Staubli VAL3: Robot_pippeting.pjx

--- Robot_pippeting.pjx ---
Parameters version=s8.8.3cs9_BS1660 stackSize=200000 millimeterUnit=true
Program file=ComPlc.pgx
Program file=Control.pgx
Program file=Emergencia.pgx
Program file=Init.pgx
Program file=Log.pgx
Program file=N10_AproBanyera.pgx
Program file=N11_Banyera.pgx
Program file=N12_AproAmpolla.pgx
Program file=N13_Ampolla.pgx
Program file=N15_AproAgafarPuntes.pgx
Program file=N16_AgafarPuntes.pgx
Program file=N17_AproTirarPuntes.pgx
Program file=N18_TirarPuntes.pgx
Program file=N1_Home.pgx
Program file=N20_AproDosi.pgx
Program file=N21_Dosi.pgx
Program file=N22_PosDosi.pgx
Program file=Principal.pgx
Program file=Safety.pgx
Program file=Supervision.pgx
Program file=start.pgx
Program file=stop.pgx
Data file=Robot_pippeting.dtx

--- Robot_pippeting.dtx ---
aio aiAngleInclinarPipieta = {link=E954DA08-7D0C-47C0-8458-4D7DB0686071}
aio aiNumAmpolla = {link=F94C03B3-E86B-41EA-9D21-23C2AFB25672}
aio aiNumBanyera = {link=3DE16CC9-CC25-4818-8F3E-A7F806CB7947}
aio aiNumPipeta = {link=5259214B-6548-4F3D-A189-73563EE6598D}
aio aiNumPlacaDosi = {link=C4FBE503-E51F-4D58-BE10-749D221ACEB2}
aio aiProgramaPlc = {link=8E5652B8-E4D3-4267-ADD0-9C5A815DF2D8}
aio aiWordComPlc = {link=5C2A04D3-4005-4B43-8647-C0FC7B49D3AE}
aio aiXOffset = {link=95067B68-557B-4170-88AF-FC9CF5B8ED7A}
aio aiYOffset = {link=396181D2-5171-4A97-9799-32514BBB5F95}
aio aiZApro = {link=2D158B67-9924-4741-B554-50FB73F41045}
aio aiZOffset = {link=7513B562-B4FE-4098-AA1C-29A8706B731C}
aio aoForceJ1 = {link=9B11B2FE-99BA-4B55-9ED8-E4037A61E514}
aio aoForceJ2 = {link=DFC528C5-C573-4C02-A89E-35D8A1151078}
aio aoForceJ3 = {link=EC117CCB-E5D8-4A5C-AB6E-61FBA1760A17}
aio aoForceJ4 = {link=24340562-5DCA-47E3-A269-832024611405}
aio aoForceJ5 = {link=DB01A7CB-9BAD-4D46-B614-A585779504D9}
aio aoForceJ6 = {link=7A496CE7-D747-4637-B99A-202C76C7E7CC}
aio aoProgramaRobot = {link=5113B9A1-604C-4D8B-9163-7217CBF800C7}
aio aoStatusRobot = {link=F45B1EFD-4428-4D7D-8172-ECCCA511584C}
aio aoTascaAlarma = {link=53CEF201-0BB5-4BE1-8271-49FFF55CF52D}
aio aoWordComRobot = {link=6DF138BB-5CBA-4ACE-9C62-0AC3DF2353CB}
aio aoWorkingMode = {link=F7E03293-48A3-4B69-9598-2FE8DDFE0186}
aio aoXActual = {link=7FC267A8-BFA4-4039-BDA4-9FB4B4F71D48}
aio aoYActual = {link=E23CA4B2-A08C-4C00-8E97-94551E73BB09}
aio aoZActual = {link=78A73075-60CA-4FDB-AFF0-231125481CE1}
aio aoZonaHome = {link=F5709703-FBB2-4816-9A2C-2FC6F0D8F434}
bool bNewLog
bool bPrimerCicle
bool bTaskDone
dio diAlarmaPlc = {link=E7921EDF-610C-4E3F-84A7-2F1F4421B713}
dio diMarxaMaquina = {link=C1F67030-A9C1-420C-9B9B-1F49F7080557}
dio diSafetyRearme = {link=5367EF22-1F58-447B-AD12-D8B84F185C6B}
dio doAlarmaColisioRobot = {link=EA8AD671-7535-4BE0-BEBB-B9246DF094E3}
dio doAlarmaTascaRobot = {link=FCAEE04F-32B9-421A-B1DD-A8CEAA94D1C9}
dio doRobotEnMoviment = {link=B70DA9EE-8DF7-4C99-91DF-7149F2D942A3}
dio doRobotHome = {link=9957E281-FF01-4081-BA5E-7A249685580C}
dio doRobotPreparat = {link=19F8D819-A10B-480E-B6CD-15D2D35E2133}
dio doTaskDone = {link=0B0F13F6-DB8F-450C-AEE5-782BE1039C53}
frame fTaula = {fatherId=world[0]}
jointRx jHome = {j1=-3.455563, j2=6.0127238, j3=105.394535, j4=0.000031955, j5=68.591721, j6=-183.446968}
mdesc mAgafarPuntes = {accel=10, vel=10, decel=10, leave=0, reach=0}
mdesc mHome = {accel=25, vel=25, decel=25, leave=0, reach=0}
mdesc mLent = {accel=25, vel=25, decel=25, leave=10, reach=10}
mdesc mMig = {accel=50, vel=50, decel=50}
mdesc mNomSpeed
num nAngleInclinarPipeta
num nInerciaEina[3 3]
  [0,0] = 0.284
  [1,1] = 0.348
  [2,2] = 0.212
num nJointForce[6]
  [0] = 1.760942
  [1] = -21.676362
  [2] = -3.171848
  [3] = 1.641233
  [4] = -2.820579
  [5] = -0.389449
num nLog
num nPesEina = 15.8
num nSeqHome
num nWordComRobot = 6190
num nXOffset
num nYOffset
num nZApro = 50
num nZOffset
pointRx pAgafarPuntes1 = {x=287.432018, y=270.157151, z=-382.0291842, rx=179.996843, ry=-0.00380694, rz=0.700516, shoulder=lefty, elbow=epositive, wrist=wpositive, fatherId=fTaula[0]}
pointRx pAgafarPuntes8 = {x=285.860304, y=302.266054, z=-361.378441, rx=179.997149, ry=-0.00370527, rz=0.700442, shoulder=lefty, elbow=epositive, wrist=wpositive, fatherId=fTaula[0]}
pointRx pAmpolla[3]
  [0] = {x=493.522667, y=144.0778037, z=-386.621607, rx=179.997388, ry=-0.00407881, rz=0.700451, shoulder=lefty, elbow=epositive, wrist=wpositive, fatherId=fTaula[0]}
  [1] = {x=493.522667, y=144.0778037, z=-386.621607, rx=179.997388, ry=-0.00407881, rz=0.700451, shoulder=lefty, elbow=epositive, wrist=wpositive, fatherId=fTaula[0]}
  [2] = {x=546.605553, y=142.888702, z=-386.0523536, rx=179.997158, ry=-0.00493572, rz=0.700473, shoulder=lefty, elbow=epositive, wrist=wpositive, fatherId=fTaula[0]}
pointRx pBanyera[3]
  [0] = {x=336.466109, y=102.428458, z=-384.993166, rx=-0.00440943, ry=-179.995824, rz=-89.890495, shoulder=lefty, elbow=epositive, wrist=wpositive, fatherId=fTaula[0]}
  [1] = {x=336.466109, y=102.428458, z=-384.993166, rx=-0.00440943, ry=-179.995824, rz=-89.890495, shoulder=lefty, elbow=epositive, wrist=wpositive, fatherId=fTaula[0]}
  [2] = {x=336.466107, y=182.839383, z=-384.995018, rx=-0.003849, ry=-179.995539, rz=-89.890699, shoulder=lefty, elbow=epositive, wrist=wpositive, fatherId=fTaula[0]}
pointRx pDosi1[4]
  [0] = {x=305.52358, y=28.950334, z=-381.105899, rx=-0.00502749, ry=-179.983412, rz=-88.969574, shoulder=lefty, elbow=epositive, wrist=wpositive, fatherId=fTaula[0]}
  [1] = {x=305.523534, y=28.950368, z=-381.105899, rx=-0.00502365, ry=-179.983406, rz=-88.969579, shoulder=lefty, elbow=epositive, wrist=wpositive, fatherId=fTaula[0]}
  [2] = {x=306.96586, y=-130.963134, z=-381.122863, rx=-0.00532463, ry=-179.983113, rz=-88.9695, shoulder=lefty, elbow=epositive, wrist=wpositive, fatherId=fTaula[0]}
  [3] = {x=307.512874, y=-290.507285, z=-381.117547, rx=-0.00478912, ry=-179.98278, rz=-88.969551, shoulder=lefty, elbow=epositive, wrist=wpositive, fatherId=fTaula[0]}
pointRx pDosi8[4]
  [0] = {x=337.355483, y=31.174712, z=-385.0727918, rx=-0.0019009, ry=-179.993411, rz=-88.962152, shoulder=lefty, elbow=epositive, wrist=wpositive, fatherId=fTaula[0]}
  [1] = {x=337.355483, y=31.174712, z=-385.0727918, rx=-0.0019009, ry=-179.993411, rz=-88.962152, shoulder=lefty, elbow=epositive, wrist=wpositive, fatherId=fTaula[0]}
  [2] = {x=338.549957, y=-128.589669, z=-385.0544196, rx=0.000914256, ry=-179.993163, rz=-88.965193, shoulder=lefty, elbow=epositive, wrist=wpositive, fatherId=fTaula[0]}
  [3] = {x=339.326592, y=-288.609993, z=-385.0722156, rx=0.00206439, ry=-179.994818, rz=-88.964134, shoulder=lefty, elbow=epositive, wrist=wpositive, fatherId=fTaula[0]}
pointRx pHereHome = {x=172.623152, y=-333.816468, z=-286.331237, rx=0.00171927, ry=-179.997666, rz=-88.962057, shoulder=lefty, elbow=epositive, wrist=wpositive, fatherId=fTaula[0]}
pointRx pHome = {x=319.622111, y=0.736493, z=-179.743756, rx=180, shoulder=lefty, elbow=epositive, wrist=wpositive, fatherId=fTaula[0]}
pointRx pTirarPuntes = {x=172.623152, y=-333.816468, z=-336.331237, rx=0.00171927, ry=-179.997666, rz=-88.962057, shoulder=lefty, elbow=epositive, wrist=wpositive, fatherId=fTaula[0]}
string sLog[50]
  [1] = "1 - Inici: HOME"
  [2] = "17 - Fi: ANAR A APRO TIRAR PUNTES"
  [3] = "17 - Inici: ANAR A APRO TIRAR PUNTES"
  [4] = "18 - Fi: ANAR A TIRAR PUNTES"
  [5] = "18 - Inici: ANAR A TIRAR PUNTES"
  [6] = "17 - Fi: ANAR A APRO TIRAR PUNTES"
  [7] = "17 - Inici: ANAR A APRO TIRAR PUNTES"
  [8] = "20 - Fi: ANAR A APRO DOSI"
  [9] = "20 - Inici: ANAR A APRO DOSI"
  [10] = "22 - Fi: ANAR A POSICIONAT DOSI"
  [11] = "22 - Inici: ANAR A POSICIONAT DOSI"
  [12] = "21 - Fi: ANAR A DOSI"
  [13] = "21 - Inici: ANAR A DOSI"
  [14] = "20 - Fi: ANAR A APRO DOSI"
  [15] = "20 - Inici: ANAR A APRO DOSI"
  [16] = "20 - Fi: ANAR A APRO DOSI"
  [17] = "20 - Inici: ANAR A APRO DOSI"
  [18] = "22 - Fi: ANAR A POSICIONAT DOSI"
  [19] = "22 - Inici: ANAR A POSICIONAT DOSI"
  [20] = "21 - Fi: ANAR A DOSI"
  [21] = "21 - Inici: ANAR A DOSI"
  [22] = "20 - Fi: ANAR A APRO DOSI"
  [23] = "20 - Inici: ANAR A APRO DOSI"
  [24] = "20 - Fi: ANAR A APRO DOSI"
  [25] = "20 - Inici: ANAR A APRO DOSI"
  [26] = "21 - Fi: ANAR A DOSI"
  [27] = "21 - Inici: ANAR A DOSI"
  [28] = "20 - Fi: ANAR A APRO DOSI"
  [29] = "20 - Inici: ANAR A APRO DOSI"
  [30] = "15 - Fi: ANAR A APRO AGAFAR PUNTES"
  [31] = "15 - Inici: ANAR A APRO AGAFAR PUNTES"
  [32] = "16 - Fi: ANAR A AGAFAR PUNTES"
  [33] = "16 - Inici: ANAR A AGAFAR PUNTES"
  [34] = "15 - Fi: ANAR A APRO AGAFAR PUNTES"
  [35] = "15 - Inici: ANAR A APRO AGAFAR PUNTES"
  [36] = "17 - Fi: ANAR A APRO TIRAR PUNTES"
  [37] = "17 - Inici: ANAR A APRO TIRAR PUNTES"
  [38] = "18 - Fi: ANAR A TIRAR PUNTES"
  [39] = "18 - Inici: ANAR A TIRAR PUNTES"
  [40] = "17 - Fi: ANAR A APRO TIRAR PUNTES"
  [41] = "17 - Inici: ANAR A APRO TIRAR PUNTES"
  [42] = "20 - Fi: ANAR A APRO DOSI"
  [43] = "20 - Inici: ANAR A APRO DOSI"
  [44] = "22 - Fi: ANAR A POSICIONAT DOSI"
  [45] = "22 - Inici: ANAR A POSICIONAT DOSI"
  [46] = "21 - Fi: ANAR A DOSI"
  [47] = "21 - Inici: ANAR A DOSI"
  [48] = "20 - Fi: ANAR A APRO DOSI"
  [49] = "20 - Inici: ANAR A APRO DOSI"
string sNewLog = "1 - Fi: HOME"
tool tToolActiva = {z=285, fatherId=flange[0]}
tool tToolPipeta1 = {z=300, fatherId=flange[0]}
tool tToolPipeta8 = {z=285, fatherId=flange[0]}
trsf trEina = {x=94.8, y=-0.4, z=220.5}

--- start.pgx ---
program start()
begin

  taskCreate "Supervision",50,Supervision()
  taskCreate "ComPlc",50,ComPlc()
  taskCreate "Init",50,Init()

  // Mostrar pantalla d'usuari
  userPage("main")
end

--- ComPlc.pgx ---
program ComPlc()
begin
  do
    // Word de vida de la comunicació entre el robot i el PLC
    if nWordComRobot>10000
      nWordComRobot=0
    endIf
    nWordComRobot=nWordComRobot+1
    aioSet(aoWordComRobot,nWordComRobot)

  until false
end

--- Control.pgx ---
program Control()
  local pointRx l_pHere
begin
  do
    // Status robot
    aioSet(aoStatusRobot,esStatus())
    aioSet(aoWorkingMode,workingMode())

    // Velocitat del robot segons hmi
    //setMonitorSpeed(aioGet(aiVelocitatRobot))

    // Donar potencia al robot
    if esStatus()==0 and diAlarmaPlc==false and isPowered()==false and workingMode()==4
      enablePower()
    endIf

    // Definir tool de treball
    if aioGet(aiNumPipeta)==2
      tToolActiva=tToolPipeta8
    else
      tToolActiva=tToolPipeta1
    endIf

    // Envelope error - Alarma possible colisió del robot
    //doAlarmaColisioRobot=$envelopeError()

    // Error "Posició cartesiana fóra de límits"
    if taskStatus("Principal")==531 or taskStatus("N1_Home")==531 or taskStatus("N10_AproBanyera")==531 or taskStatus("N11_Banyera")==531 or taskStatus("N15_AproAgafarPuntes")==531 or taskStatus("N16_AgafarPuntes")==531 or taskStatus("N17_AproTirarPuntes")==531 or taskStatus("N18_TirarPuntes")==531 or taskStatus("N20_AproDosi")==531 or taskStatus("N21_Dosi")==531 or taskStatus("N22_PosDosi")==531 or taskStatus("N12_AproAmpolla")==531 or taskStatus("N13_Ampolla")==531
      aioSet(aoTascaAlarma,aioGet(aoProgramaRobot))
      doAlarmaTascaRobot=true
    else
      doAlarmaTascaRobot=false
    endIf

    // Enviar al PLC la força de cada motor del robot (Nm)
    getJointForce(nJointForce)
    aioSet(aoForceJ1,nJointForce[0])
    aioSet(aoForceJ2,nJointForce[1])
    aioSet(aoForceJ3,nJointForce[2])
    aioSet(aoForceJ4,nJointForce[3])
    aioSet(aoForceJ5,nJointForce[4])
    aioSet(aoForceJ6,nJointForce[5])

    // Enviar al PLC la posició actual del robot
    l_pHere=here(tToolActiva,world)
    aioSet(aoXActual,l_pHere.trsf.x)
    aioSet(aoYActual,l_pHere.trsf.y)
    aioSet(aoZActual,l_pHere.trsf.z)

  until false
end

--- Emergencia.pgx ---
program Emergencia()
begin

  do
    if diAlarmaPlc==true

      taskKill("Principal")
      taskKill("N1_Home")
      taskKill("N10_AproBanyera")
      taskKill("N11_Banyera")
      taskKill("N12_AproAmpolla")
      taskKill("N13_Ampolla")
      taskKill("N15_AproAgafarPuntes")
      taskKill("N16_AgafarPuntes")
      taskKill("N17_AproTirarPuntes")
      taskKill("N18_TirarPuntes")
      taskKill("N20_AproDosi")
      taskKill("N21_Dosi")
      taskKill("N22_PosDosi")


      resetMotion()
      //Reset variables
      doRobotHome=false
      doRobotEnMoviment=false

      doAlarmaColisioRobot=false
      doTaskDone=false

      bTaskDone=false
      bPrimerCicle=false
      nSeqHome=0
      aioSet(aoProgramaRobot,0)
      aioSet(aoZonaHome,0)

      wait(diAlarmaPlc==false)

      taskCreate "Principal",50,Principal()
    endIf
    delay(0)
  until false


end

--- Init.pgx ---
program Init()
begin


  // Inicialització de variables
  doRobotHome=false
  doRobotEnMoviment=false
  doRobotPreparat=false
  doAlarmaColisioRobot=false
  doAlarmaTascaRobot=false
  doTaskDone=false
  bTaskDone=false
  bPrimerCicle=false
  bNewLog=false
  sLog=""
  nSeqHome=0
  aioSet(aoProgramaRobot,0)
  aioSet(aoZonaHome,0)
  nAngleInclinarPipeta=0

  //  // Definir l'eina (valores de inercia en kg·m2)
  nInerciaEina[0,0]=0.284
  nInerciaEina[0,1]=0
  nInerciaEina[0,2]=0
  nInerciaEina[1,0]=0
  nInerciaEina[1,1]=0.348
  nInerciaEina[1,2]=0
  nInerciaEina[2,0]=0
  nInerciaEina[2,1]=0
  nInerciaEina[2,2]=0.212
  trEina={94.8,-0.4,220.5,0,0,0}
  nPesEina=15.8
  setPayload(flange,nPesEina,trEina,nInerciaEina)


  doRobotPreparat=true

  taskCreate "Control",50,Control()
  taskCreate "Log",50,Log()
  taskCreate "Safety",50,Safety()
  taskCreate "Principal",50,Principal()
  taskCreate "Emergencia",2,Emergencia()

end

--- Log.pgx ---
program Log()
begin
  do
    // Registrar un nou event al logger
    if bNewLog==true
      // Desplaçar registre d'events
      for nLog=49 to 1 step -1
        sLog[nLog]=sLog[nLog-1]
      endFor
      // Afegir nou event
      sLog[0]=sNewLog
      bNewLog=false
    endIf

  until false
end

--- N10_AproBanyera.pgx ---
program N10_AproBanyera()
  local pointRx l_pAproBanyera
begin

  // Anar a l'aproximació del punt d'agafar líquid de la banyera
  l_pAproBanyera=pBanyera[aioGet(aiNumBanyera)]
  l_pAproBanyera.trsf.x=l_pAproBanyera.trsf.x+nXOffset
  l_pAproBanyera.trsf.y=l_pAproBanyera.trsf.y+nYOffset
  l_pAproBanyera.trsf.z=l_pAproBanyera.trsf.z+nZOffset

  if nZApro>0
    l_pAproBanyera.trsf.z=l_pAproBanyera.trsf.z+nZApro
  else
    l_pAproBanyera.trsf.z=l_pAproBanyera.trsf.z+100
  endIf

  movel(l_pAproBanyera,tToolActiva,mLent)
  waitEndMove()

  bTaskDone=true
end

--- N11_Banyera.pgx ---
program N11_Banyera()
  local pointRx l_pBanyera
begin

  // Anar al punt de la banyera
  l_pBanyera=pBanyera[aioGet(aiNumBanyera)]
  l_pBanyera.trsf.x=l_pBanyera.trsf.x+nXOffset
  l_pBanyera.trsf.y=l_pBanyera.trsf.y+nYOffset
  l_pBanyera.trsf.z=l_pBanyera.trsf.z+nZOffset
  movel(l_pBanyera,tToolActiva,mLent)
  waitEndMove()

  bTaskDone=true
end

--- N12_AproAmpolla.pgx ---
program N12_AproAmpolla()
  local pointRx l_pAproAmpolla
begin

  // Anar a l'aproximació del punt d'agafar líquid de l'ampolla
  l_pAproAmpolla=pAmpolla[aioGet(aiNumAmpolla)]
  l_pAproAmpolla.trsf.x=l_pAproAmpolla.trsf.x+nXOffset
  l_pAproAmpolla.trsf.y=l_pAproAmpolla.trsf.y+nYOffset
  l_pAproAmpolla.trsf.z=l_pAproAmpolla.trsf.z+nZOffset

  if nZApro>0
    l_pAproAmpolla.trsf.z=l_pAproAmpolla.trsf.z+nZApro
  else
    l_pAproAmpolla.trsf.z=l_pAproAmpolla.trsf.z+100
  endIf

  movel(l_pAproAmpolla,tToolActiva,mLent)
  waitEndMove()

  bTaskDone=true
end

--- N13_Ampolla.pgx ---
program N13_Ampolla()
  local pointRx l_pAmpolla
begin

  // Anar al punt de l'ampolla
  l_pAmpolla=pAmpolla[aioGet(aiNumAmpolla)]
  l_pAmpolla.trsf.x=l_pAmpolla.trsf.x+nXOffset
  l_pAmpolla.trsf.y=l_pAmpolla.trsf.y+nYOffset
  l_pAmpolla.trsf.z=l_pAmpolla.trsf.z+nZOffset
  movel(l_pAmpolla,tToolActiva,mLent)
  waitEndMove()

  bTaskDone=true
end

--- N15_AproAgafarPuntes.pgx ---
program N15_AproAgafarPuntes()
  local pointRx l_pAproAgafarPuntes
begin

  // Anar a l'aproximació del punt d'agafar puntes
  if aioGet(aiNumPipeta)==2
    l_pAproAgafarPuntes=pAgafarPuntes8
  else
    l_pAproAgafarPuntes=pAgafarPuntes1
  endIf

  l_pAproAgafarPuntes.trsf.x=l_pAproAgafarPuntes.trsf.x+nXOffset
  l_pAproAgafarPuntes.trsf.y=l_pAproAgafarPuntes.trsf.y+nYOffset
  l_pAproAgafarPuntes.trsf.z=l_pAproAgafarPuntes.trsf.z+nZOffset

  if nZApro>0
    l_pAproAgafarPuntes.trsf.z=l_pAproAgafarPuntes.trsf.z+nZApro
  else
    l_pAproAgafarPuntes.trsf.z=l_pAproAgafarPuntes.trsf.z+100
  endIf

  movel(l_pAproAgafarPuntes,tToolActiva,mLent)
  waitEndMove()

  bTaskDone=true
end

--- N16_AgafarPuntes.pgx ---
program N16_AgafarPuntes()
  local pointRx l_pAgafarPuntes
  local pointRx l_pAgafarPuntesRapid
begin

  // Anar al punt de la banyera
  if aioGet(aiNumPipeta)==2
    l_pAgafarPuntes=pAgafarPuntes8
  else
    l_pAgafarPuntes=pAgafarPuntes1
  endIf

  l_pAgafarPuntes.trsf.x=l_pAgafarPuntes.trsf.x+nXOffset
  l_pAgafarPuntes.trsf.y=l_pAgafarPuntes.trsf.y+nYOffset
  l_pAgafarPuntes.trsf.z=l_pAgafarPuntes.trsf.z+nZOffset
  l_pAgafarPuntesRapid=l_pAgafarPuntes
  l_pAgafarPuntesRapid.trsf.z=l_pAgafarPuntesRapid.trsf.z+20
  movel(l_pAgafarPuntesRapid,tToolActiva,mLent)
  waitEndMove()
  movel(l_pAgafarPuntes,tToolActiva,mAgafarPuntes)
  waitEndMove()

  bTaskDone=true
end

--- N17_AproTirarPuntes.pgx ---
program N17_AproTirarPuntes()
  local pointRx l_pAproTirarPuntes
begin

  // Anar a l'aproximació del punt de tirar puntes
  l_pAproTirarPuntes=pTirarPuntes
  l_pAproTirarPuntes.trsf.x=l_pAproTirarPuntes.trsf.x+nXOffset
  l_pAproTirarPuntes.trsf.y=l_pAproTirarPuntes.trsf.y+nYOffset
  l_pAproTirarPuntes.trsf.z=l_pAproTirarPuntes.trsf.z+nZOffset

  if nZApro>0
    l_pAproTirarPuntes.trsf.z=l_pAproTirarPuntes.trsf.z+nZApro
  else
    l_pAproTirarPuntes.trsf.z=l_pAproTirarPuntes.trsf.z+50
  endIf

  movel(l_pAproTirarPuntes,tToolActiva,mLent)
  waitEndMove()

  bTaskDone=true
end

--- N18_TirarPuntes.pgx ---
program N18_TirarPuntes()
  local pointRx l_pTirarPuntes
begin

  // Anar al punt de tirar puntes
  l_pTirarPuntes=pTirarPuntes
  l_pTirarPuntes.trsf.x=l_pTirarPuntes.trsf.x+nXOffset
  l_pTirarPuntes.trsf.y=l_pTirarPuntes.trsf.y+nYOffset
  l_pTirarPuntes.trsf.z=l_pTirarPuntes.trsf.z+nZOffset
  movel(l_pTirarPuntes,tToolActiva,mLent)
  waitEndMove()

  bTaskDone=true
end

--- N1_Home.pgx ---
program N1_Home()
  local pointRx l_pHere
begin
  do

    switch nSeqHome

      // Inici de la seqüència
      case 0
        // Anar a home
        doRobotHome=false
        doRobotEnMoviment=true
        aioSet(aoZonaHome,0)
        waitEndMove()
        // Comprovar a quina posició es troba el robot
        l_pHere=here(tToolActiva,fTaula)
        pHereHome=l_pHere
        nSeqHome=10
      break

      // Pujar verticalment fins a una cota segura en Z
      case 10
        if l_pHere.trsf.z<pHome.trsf.z
          l_pHere.trsf.z=pHome.trsf.z
          movel(l_pHere,tToolActiva,mHome)
          waitEndMove()
          nSeqHome=20
        else
          nSeqHome=20
        endIf
      break

      // Comprovar on es troba el robot
      case 20
        // Ja està en posició de Home
        aioSet(aoZonaHome,99)
        nSeqHome=1000
      break

      // Fi del HOME
      case 1000
        movel(pHome,tToolActiva,mHome)
        waitEndMove()
        doRobotHome=true
        doRobotEnMoviment=false
        bTaskDone=true
        nSeqHome=1001
      break
    endSwitch
  until nSeqHome==1001
end

--- N20_AproDosi.pgx ---
program N20_AproDosi()
  local pointRx l_pAproDosi
begin

  // Anar a l'aproximació vertical de dosificar placa
  if aioGet(aiNumPipeta)==2
    l_pAproDosi=pDosi8[aioGet(aiNumPlacaDosi)]
  else
    l_pAproDosi=pDosi1[aioGet(aiNumPlacaDosi)]
  endIf

  l_pAproDosi.trsf.x=l_pAproDosi.trsf.x+nXOffset
  l_pAproDosi.trsf.y=l_pAproDosi.trsf.y+nYOffset
  l_pAproDosi.trsf.z=l_pAproDosi.trsf.z+nZOffset

  if nZApro>0
    l_pAproDosi.trsf.z=l_pAproDosi.trsf.z+nZApro
  else
    l_pAproDosi.trsf.z=l_pAproDosi.trsf.z+25
  endIf

  l_pAproDosi.trsf.rx=l_pAproDosi.trsf.rx+aioGet(aiAngleInclinarPipieta)

  movel(l_pAproDosi,tToolActiva,mLent)
  waitEndMove()

  bTaskDone=true
end

--- N21_Dosi.pgx ---
program N21_Dosi()
  local pointRx l_pDosi
begin

  // Anar al punt de dosificar placa
  if aioGet(aiNumPipeta)==2
    l_pDosi=pDosi8[aioGet(aiNumPlacaDosi)]
  else
    l_pDosi=pDosi1[aioGet(aiNumPlacaDosi)]
  endIf
  l_pDosi.trsf.x=l_pDosi.trsf.x+nXOffset
  l_pDosi.trsf.y=l_pDosi.trsf.y+nYOffset
  l_pDosi.trsf.z=l_pDosi.trsf.z+nZOffset
  l_pDosi.trsf.rx=l_pDosi.trsf.rx+aioGet(aiAngleInclinarPipieta)

  movel(l_pDosi,tToolActiva,mLent)
  waitEndMove()

  bTaskDone=true
end

--- N22_PosDosi.pgx ---
program N22_PosDosi()
  local pointRx l_pDosi
begin

  // Moure puntes per treure les gotes
  l_pDosi=here(tToolActiva,fTaula)
  l_pDosi.trsf.x=l_pDosi.trsf.x+nXOffset
  l_pDosi.trsf.y=l_pDosi.trsf.y+nYOffset
  l_pDosi.trsf.z=l_pDosi.trsf.z+nZOffset
  movel(l_pDosi,tToolActiva,mLent)
  waitEndMove()

  bTaskDone=true
end

--- Principal.pgx ---
program Principal()
begin
  do

    // Esperar aiProgramaPlc <> 0
    do
      delay(0)
    until (aioGet(aiProgramaPlc)!=0)

    // Processar X,Y,Z offset posició
    nXOffset=aioGet(aiXOffset)/100
    nYOffset=aioGet(aiYOffset)/100
    nZOffset=aioGet(aiZOffset)/100
    nZApro=aioGet(aiZApro)

    bTaskDone=false
    doTaskDone=false
    doRobotEnMoviment=true
    doRobotHome=false
    // Cridar programa corresponent
    switch aioGet(aiProgramaPlc)
      // 1: HOME
      case 1
        wait(bNewLog==false)
        sNewLog="1 - Inici: HOME"
        bNewLog=true
        nSeqHome=0
        aioSet(aoProgramaRobot,1)
        taskCreate "N1_Home",50,N1_Home()
        wait(bTaskDone==true)
        wait(aioGet(aiProgramaPlc)==0)
        aioSet(aoProgramaRobot,0)
        doTaskDone=true
        wait(bNewLog==false)
        sNewLog="1 - Fi: HOME"
        bNewLog=true
      break

      // 10: ANAR A APRO BANYERA
      case 10
        wait(bNewLog==false)
        sNewLog="10 - Inici: ANAR A APRO BANYERA"
        bNewLog=true
        aioSet(aoProgramaRobot,10)
        taskCreate "N10_AproBanyera",50,N10_AproBanyera()
        wait(bTaskDone==true)
        wait(aioGet(aiProgramaPlc)==0)
        aioSet(aoProgramaRobot,0)
        doTaskDone=true
        wait(bNewLog==false)
        sNewLog="10 - Fi: ANAR A APRO BANYERA"
        bNewLog=true
      break

      // 11: ANAR A BANYERA
      case 11
        wait(bNewLog==false)
        sNewLog="11 - Inici: ANAR A BANYERA"
        bNewLog=true
        aioSet(aoProgramaRobot,11)
        taskCreate "N11_Banyera",50,N11_Banyera()
        wait(bTaskDone==true)
        wait(aioGet(aiProgramaPlc)==0)
        aioSet(aoProgramaRobot,0)
        doTaskDone=true
        wait(bNewLog==false)
        sNewLog="11 - Fi: ANAR A BANYERA"
        bNewLog=true
      break

      // 12: ANAR A APRO AMPOLLA
      case 12
        wait(bNewLog==false)
        sNewLog="12 - Inici: ANAR A APRO AMPOLLA"
        bNewLog=true
        aioSet(aoProgramaRobot,12)
        taskCreate "N12_AproAmpolla",50,N12_AproAmpolla()
        wait(bTaskDone==true)
        wait(aioGet(aiProgramaPlc)==0)
        aioSet(aoProgramaRobot,0)
        doTaskDone=true
        wait(bNewLog==false)
        sNewLog="12 - Fi: ANAR A APRO AMPOLLA"
        bNewLog=true
      break

      // 13: ANAR A AMPOLLA
      case 13
        wait(bNewLog==false)
        sNewLog="13 - Inici: ANAR A AMPOLLA"
        bNewLog=true
        aioSet(aoProgramaRobot,13)
        taskCreate "N13_Ampolla",50,N13_Ampolla()
        wait(bTaskDone==true)
        wait(aioGet(aiProgramaPlc)==0)
        aioSet(aoProgramaRobot,0)
        doTaskDone=true
        wait(bNewLog==false)
        sNewLog="13 - Fi: ANAR A AMPOLLA"
        bNewLog=true
      break

      // 15: ANAR A APRO AGAFAR PUNTES
      case 15
        wait(bNewLog==false)
        sNewLog="15 - Inici: ANAR A APRO AGAFAR PUNTES"
        bNewLog=true
        aioSet(aoProgramaRobot,15)
        taskCreate "N15_AproAgafarPuntes",50,N15_AproAgafarPuntes()
        wait(bTaskDone==true)
        wait(aioGet(aiProgramaPlc)==0)
        aioSet(aoProgramaRobot,0)
        doTaskDone=true
        wait(bNewLog==false)
        sNewLog="15 - Fi: ANAR A APRO AGAFAR PUNTES"
        bNewLog=true
      break

      // 16: ANAR A AGAFAR PUNTES
      case 16
        wait(bNewLog==false)
        sNewLog="16 - Inici: ANAR A AGAFAR PUNTES"
        bNewLog=true
        aioSet(aoProgramaRobot,16)
        taskCreate "N16_AgafarPuntes",50,N16_AgafarPuntes()
        wait(bTaskDone==true)
        wait(aioGet(aiProgramaPlc)==0)
        aioSet(aoProgramaRobot,0)
        doTaskDone=true
        wait(bNewLog==false)
        sNewLog="16 - Fi: ANAR A AGAFAR PUNTES"
        bNewLog=true
      break

      // 17: ANAR A APRO TIRAR PUNTES
      case 17
        wait(bNewLog==false)
        sNewLog="17 - Inici: ANAR A APRO TIRAR PUNTES"
        bNewLog=true
        aioSet(aoProgramaRobot,17)
        taskCreate "N17_AproTirarPuntes",50,N17_AproTirarPuntes()
        wait(bTaskDone==true)
        wait(aioGet(aiProgramaPlc)==0)
        aioSet(aoProgramaRobot,0)
        doTaskDone=true
        wait(bNewLog==false)
        sNewLog="17 - Fi: ANAR A APRO TIRAR PUNTES"
        bNewLog=true
      break

      // 18: ANAR A TIRAR PUNTES
      case 18
        wait(bNewLog==false)
        sNewLog="18 - Inici: ANAR A TIRAR PUNTES"
        bNewLog=true
        aioSet(aoProgramaRobot,18)
        taskCreate "N18_TirarPuntes",50,N18_TirarPuntes()
        wait(bTaskDone==true)
        wait(aioGet(aiProgramaPlc)==0)
        aioSet(aoProgramaRobot,0)
        doTaskDone=true
        wait(bNewLog==false)
        sNewLog="18 - Fi: ANAR A TIRAR PUNTES"
        bNewLog=true
      break

      // 20: ANAR A APRO DOSI
      case 20
        wait(bNewLog==false)
        sNewLog="20 - Inici: ANAR A APRO DOSI"
        bNewLog=true
        aioSet(aoProgramaRobot,20)
        taskCreate "N20_AproDosi",50,N20_AproDosi()
        wait(bTaskDone==true)
        wait(aioGet(aiProgramaPlc)==0)
        aioSet(aoProgramaRobot,0)
        doTaskDone=true
        wait(bNewLog==false)
        sNewLog="20 - Fi: ANAR A APRO DOSI"
        bNewLog=true
      break

      // 21: ANAR A DOSI
      case 21
        wait(bNewLog==false)
        sNewLog="21 - Inici: ANAR A DOSI"
        bNewLog=true
        aioSet(aoProgramaRobot,21)
        taskCreate "N21_Dosi",50,N21_Dosi()
        wait(bTaskDone==true)
        wait(aioGet(aiProgramaPlc)==0)
        aioSet(aoProgramaRobot,0)
        doTaskDone=true
        wait(bNewLog==false)
        sNewLog="21 - Fi: ANAR A DOSI"
        bNewLog=true
      break

      // 22: ANAR A POSICIONAT DOSI
      case 22
        wait(bNewLog==false)
        sNewLog="22 - Inici: ANAR A POSICIONAT DOSI"
        bNewLog=true
        aioSet(aoProgramaRobot,22)
        taskCreate "N22_PosDosi",50,N22_PosDosi()
        wait(bTaskDone==true)
        wait(aioGet(aiProgramaPlc)==0)
        aioSet(aoProgramaRobot,0)
        doTaskDone=true
        wait(bNewLog==false)
        sNewLog="22 - Fi: ANAR A POSICIONAT DOSI"
        bNewLog=true
      break


    endSwitch


  until false

end

--- Safety.pgx ---
program Safety()
begin
  do

    // Rearme del safety
    if diSafetyRearme==true and esStatus()==1
      setSafetyRestart()
    endIf


  until false
end

--- Supervision.pgx ---
program Supervision()
begin
  do


    if ioStatus(aiWordComPlc)>=0
      if taskStatus("ComPlc")==125
        taskResume("ComPlc",1)
      endIf
      if taskStatus("Init")==125
        taskResume("Init",1)
      endIf

      if taskStatus("Control")==125
        taskResume("Control",1)
      endIf

      if taskStatus("Emergencia")==125
        taskResume("Emergencia",1)
      endIf

      if taskStatus("Home")==125
        taskResume("Home",1)
      endIf

      if taskStatus("Principal")==125
        taskResume("Principal",1)
      endIf

      if taskStatus("Safety")==125
        taskResume("Safety",1)
      endIf

      if taskStatus("N10_AproBanyera")==125
        taskResume("N10_AnarBanyera",1)
      endIf

      if taskStatus("N11_Banyera")==125
        taskResume("N11_Banyera",1)
      endIf

      if taskStatus("N12_AproAmpolla")==125
        taskResume("N12_AproAmpolla",1)
      endIf

      if taskStatus("N13_Ampolla")==125
        taskResume("N13_Ampolla",1)
      endIf

      if taskStatus("N15_AproAgafarPuntes")==125
        taskResume("N15_AproAgafarPuntes",1)
      endIf

      if taskStatus("N16_AgafarPuntes")==125
        taskResume("N16_AgafarPuntes",1)
      endIf

      if taskStatus("N17_AproTirarPuntes")==125
        taskResume("N17_AproTirarPuntes",1)
      endIf

      if taskStatus("N18_TirarPuntes")==125
        taskResume("N18_TirarPuntes",1)
      endIf

      if taskStatus("N20_AproDosi")==125
        taskResume("N20_AproDosi",1)
      endIf

      if taskStatus("N21_Dosi")==125
        taskResume("N21_Dosi",1)
      endIf

      if taskStatus("N22_PosDosi")==125
        taskResume("N22_PosiDosi",1)
      endIf

    endIf
  until false
end
